(* IEC 61131-3 sources: smart-traffic-light/src/FunctionBlocks, 5 files *)

(* ---- PedestrianLight.st ---- *)
(* PedestrianLight Function Block
   Extends TrafficLight with pedestrian signal logic.
   Manages WALK/DONT_WALK/FLASHING states coordinated with the traffic signal. *)

FUNCTION_BLOCK PedestrianLight EXTENDS TrafficLight
  VAR_INPUT
    walkRequest  : BOOL := FALSE;
    walkDuration : TIME := T#20s;
  END_VAR

  VAR_OUTPUT
    pedestrianState : PedestrianState := PedestrianState.DONT_WALK;
    walkLight       : BOOL := FALSE;
    dontWalkLight   : BOOL := TRUE;
  END_VAR

  VAR
    walkTimer      : TON;
    flashTimer     : TON;
    flashCount     : INT := 0;
    maxFlashes     : INT := 5;
    flashOn        : BOOL := FALSE;
  END_VAR

  METHOD PUBLIC OVERRIDE GetState : TrafficState
    GetState := currentState;
  END_METHOD

  METHOD PUBLIC IsWalking : BOOL
    IsWalking := (pedestrianState = PedestrianState.WALK);
  END_METHOD

  METHOD PUBLIC RequestWalk : BOOL
    walkRequest := TRUE;
    RequestWalk := TRUE;
  END_METHOD

  (* Execute parent TrafficLight state machine first *)
  SUPER^();

  (* Pedestrian signal logic coordinated with traffic state *)
  IF currentState = TrafficState.RED AND walkRequest THEN
    (* Safe to walk when traffic is RED *)
    IF pedestrianState = PedestrianState.DONT_WALK THEN
      pedestrianState := PedestrianState.WALK;
      flashCount := 0;
    END_IF;

    walkTimer(IN := (pedestrianState = PedestrianState.WALK), PT := walkDuration);

    IF walkTimer.Q THEN
      pedestrianState := PedestrianState.FLASHING;
      walkTimer(IN := FALSE, PT := walkDuration);
    END_IF;

    (* Flashing phase before switching to DONT_WALK *)
    IF pedestrianState = PedestrianState.FLASHING THEN
      flashTimer(IN := TRUE, PT := T#500ms);
      IF flashTimer.Q THEN
        flashCount := flashCount + 1;
        flashOn := NOT flashOn;
        flashTimer(IN := FALSE, PT := T#500ms);
        flashTimer(IN := TRUE, PT := T#500ms);
      END_IF;

      IF flashCount >= maxFlashes THEN
        pedestrianState := PedestrianState.DONT_WALK;
        walkRequest := FALSE;
        flashCount := 0;
        flashOn := FALSE;
      END_IF;
    END_IF;
  ELSE
    (* Not safe or not requested — reset to DONT_WALK *)
    IF currentState <> TrafficState.RED THEN
      walkRequest := FALSE;
    END_IF;
    pedestrianState := PedestrianState.DONT_WALK;
    flashCount := 0;
    flashOn := FALSE;
    (* Reset timers to prevent stale state on next walk cycle *)
    walkTimer(IN := FALSE, PT := walkDuration);
    flashTimer(IN := FALSE, PT := T#500ms);
  END_IF;

  (* Update pedestrian signal outputs *)
  walkLight := (pedestrianState = PedestrianState.WALK) OR
               (pedestrianState = PedestrianState.FLASHING AND flashOn);
  dontWalkLight := (pedestrianState = PedestrianState.DONT_WALK) OR
                   (pedestrianState = PedestrianState.FLASHING AND NOT flashOn);
END_FUNCTION_BLOCK

(* ---- TrafficLight.st ---- *)
(* TrafficLight Function Block
   State machine for a standard 3-phase traffic signal.
   Cycles: RED -> GREEN -> YELLOW -> RED
   Supports night mode with flashing yellow. *)

FUNCTION_BLOCK TrafficLight IMPLEMENTS IControllable
  VAR_INPUT
    active    : BOOL := TRUE;
    timing    : PhaseTiming;
    nightMode : BOOL := FALSE;
  END_VAR

  VAR_OUTPUT
    currentState : TrafficState := TrafficState.RED;
    redLight     : BOOL := TRUE;
    yellowLight  : BOOL := FALSE;
    greenLight   : BOOL := FALSE;
  END_VAR

  VAR
    phaseTimer      : TON;
    flashTimer      : TON;
    currentDuration : TIME;
    flashOn         : BOOL := FALSE;
  END_VAR

  METHOD PUBLIC GetState : TrafficState
    GetState := currentState;
  END_METHOD

  METHOD PUBLIC IsGreen : BOOL
    IsGreen := (currentState = TrafficState.GREEN);
  END_METHOD

  METHOD PUBLIC IsRed : BOOL
    IsRed := (currentState = TrafficState.RED);
  END_METHOD

  METHOD PUBLIC IsNightMode : BOOL
    IsNightMode := nightMode;
  END_METHOD

  (* IControllable interface methods *)
  METHOD PUBLIC Enable : BOOL
    active := TRUE;
    Enable := TRUE;
  END_METHOD

  METHOD PUBLIC Disable : BOOL
    active := FALSE;
    Disable := TRUE;
  END_METHOD

  METHOD PUBLIC IsEnabled : BOOL
    IsEnabled := active;
  END_METHOD

  METHOD PUBLIC GetStatus : INT
    (* Status codes: 0=disabled, 1=RED, 2=GREEN, 3=YELLOW, 4=night mode *)
    IF NOT active THEN
      GetStatus := 0;
    ELSIF nightMode THEN
      GetStatus := 4;
    ELSIF currentState = TrafficState.RED THEN
      GetStatus := 1;
    ELSIF currentState = TrafficState.GREEN THEN
      GetStatus := 2;
    ELSE
      GetStatus := 3;
    END_IF;
  END_METHOD

  IF nightMode THEN
    (* Night mode: flash yellow at 1Hz *)
    flashTimer(IN := TRUE, PT := T#500ms);
    IF flashTimer.Q THEN
      flashOn := NOT flashOn;
      flashTimer(IN := FALSE, PT := T#500ms);
      flashTimer(IN := TRUE, PT := T#500ms);
    END_IF;

    redLight    := FALSE;
    yellowLight := flashOn;
    greenLight  := FALSE;
    currentState := TrafficState.YELLOW;
  ELSE
    (* Normal operation *)
    flashOn := FALSE;

    (* Determine the duration for the current phase *)
    CASE currentState OF
      TrafficState.RED:
        currentDuration := timing.redDuration;
      TrafficState.GREEN:
        currentDuration := timing.greenDuration;
      TrafficState.YELLOW:
        currentDuration := timing.yellowDuration;
    END_CASE;

    (* Run the phase timer *)
    phaseTimer(IN := active, PT := currentDuration);

    (* Transition to the next state when timer expires *)
    IF phaseTimer.Q THEN
      CASE currentState OF
        TrafficState.RED:
          currentState := TrafficState.GREEN;
        TrafficState.GREEN:
          currentState := TrafficState.YELLOW;
        TrafficState.YELLOW:
          currentState := TrafficState.RED;
      END_CASE;
      (* Reset timer for next phase *)
      phaseTimer(IN := FALSE, PT := currentDuration);
      phaseTimer(IN := active, PT := currentDuration);
    END_IF;

    (* Update output lights based on current state *)
    redLight    := (currentState = TrafficState.RED);
    yellowLight := (currentState = TrafficState.YELLOW);
    greenLight  := (currentState = TrafficState.GREEN);
  END_IF;
END_FUNCTION_BLOCK

(* ---- TrafficLogger.st ---- *)
(* TrafficLogger Function Block
   Maintains a circular buffer of state transition log entries.
   Uses dynamic memory allocation for the log buffer. *)

FUNCTION_BLOCK TrafficLogger
  VAR_INPUT
    bufferSize : INT := 20;
  END_VAR

  VAR_OUTPUT
    entryCount : INT := 0;
    isFull     : BOOL := FALSE;
  END_VAR

  VAR
    logBuffer    : POINTER TO LogEntry;
    writeIndex   : INT := 0;
    initialized  : BOOL := FALSE;
    totalEntries : DINT := 0;
  END_VAR

  METHOD PUBLIC Initialize : BOOL
    IF NOT initialized THEN
      logBuffer := __NEW(LogEntry, bufferSize);
      initialized := TRUE;
      Initialize := TRUE;
    ELSE
      Initialize := FALSE;
    END_IF;
  END_METHOD

  METHOD PUBLIC Cleanup : BOOL
    IF initialized THEN
      __DELETE(logBuffer);
      initialized := FALSE;
      entryCount := 0;
      writeIndex := 0;
      totalEntries := 0;
      isFull := FALSE;
      Cleanup := TRUE;
    ELSE
      Cleanup := FALSE;
    END_IF;
  END_METHOD

  METHOD PUBLIC LogTransition : BOOL
    VAR_INPUT
      fromState : TrafficState;
      toState   : TrafficState;
      time      : TIME;
    END_VAR

    IF NOT initialized THEN
      LogTransition := FALSE;
      RETURN;
    END_IF;

    logBuffer[writeIndex].previousState := fromState;
    logBuffer[writeIndex].newState := toState;
    logBuffer[writeIndex].timestamp := time;

    writeIndex := writeIndex + 1;
    IF writeIndex >= bufferSize THEN
      writeIndex := 0;
      isFull := TRUE;
    END_IF;

    totalEntries := totalEntries + 1;

    IF entryCount < bufferSize THEN
      entryCount := entryCount + 1;
    END_IF;

    LogTransition := TRUE;
  END_METHOD

  METHOD PUBLIC GetTotalTransitions : DINT
    GetTotalTransitions := totalEntries;
  END_METHOD
END_FUNCTION_BLOCK

(* ---- TurnSignalLight.st ---- *)
(* TurnSignalLight Function Block
   Extends TrafficLight with a dedicated turn signal arrow.
   The turn arrow activates during the RED-to-GREEN transition. *)

FUNCTION_BLOCK TurnSignalLight EXTENDS TrafficLight
  VAR_INPUT
    turnEnabled   : BOOL := TRUE;
    turnDuration  : TIME := T#10s;
  END_VAR

  VAR_OUTPUT
    turnArrowOn   : BOOL := FALSE;
    turnDirection : INT := 0;   (* 0=none, 1=left, 2=right *)
  END_VAR

  VAR
    turnTimer    : TON;
    turnActive   : BOOL := FALSE;
    prevState    : TrafficState := TrafficState.RED;
  END_VAR

  METHOD PUBLIC SetLeftTurn : BOOL
    turnDirection := 1;
    SetLeftTurn := TRUE;
  END_METHOD

  METHOD PUBLIC SetRightTurn : BOOL
    turnDirection := 2;
    SetRightTurn := TRUE;
  END_METHOD

  METHOD PUBLIC IsTurnActive : BOOL
    IsTurnActive := turnArrowOn;
  END_METHOD

  (* Run parent TrafficLight state machine first *)
  SUPER^();

  (* Detect RED-to-GREEN transition to activate turn signal *)
  IF prevState = TrafficState.RED AND currentState = TrafficState.GREEN THEN
    IF turnEnabled AND turnDirection > 0 THEN
      turnActive := TRUE;
    END_IF;
  END_IF;

  (* Run turn signal timer *)
  turnTimer(IN := turnActive, PT := turnDuration);
  IF turnTimer.Q THEN
    turnActive := FALSE;
    turnTimer(IN := FALSE, PT := turnDuration);
  END_IF;

  (* Turn off arrow when not in GREEN phase *)
  IF currentState <> TrafficState.GREEN THEN
    turnActive := FALSE;
  END_IF;

  turnArrowOn := turnActive;
  prevState := currentState;
END_FUNCTION_BLOCK

(* ---- VehicleDetector.st ---- *)
(* VehicleDetector Function Block
   Detects vehicles using a sensor input and maintains a detection history
   buffer allocated with dynamic memory. *)

FUNCTION_BLOCK VehicleDetector
  VAR_INPUT
    sensorInput   : BOOL := FALSE;
    maxHistory    : INT := 10;
  END_VAR

  VAR_OUTPUT
    vehicleCount  : INT := 0;
    isOccupied    : BOOL := FALSE;
    lastDetected  : TIME := T#0s;
  END_VAR

  VAR
    prevSensor     : BOOL := FALSE;
    historyBuffer  : POINTER TO INT;
    historySize    : INT := 0;
    initialized    : BOOL := FALSE;
    currentTime    : TIME := T#0s;
  END_VAR

  METHOD PUBLIC Initialize : BOOL
    IF NOT initialized THEN
      historyBuffer := __NEW(INT, maxHistory);
      initialized := TRUE;
      Initialize := TRUE;
    ELSE
      Initialize := FALSE;
    END_IF;
  END_METHOD

  METHOD PUBLIC Cleanup : BOOL
    IF initialized THEN
      __DELETE(historyBuffer);
      initialized := FALSE;
      historySize := 0;
      Cleanup := TRUE;
    ELSE
      Cleanup := FALSE;
    END_IF;
  END_METHOD

  METHOD PUBLIC GetDetectionCount : INT
    GetDetectionCount := vehicleCount;
  END_METHOD

  METHOD PUBLIC Reset : BOOL
    vehicleCount := 0;
    historySize := 0;
    isOccupied := FALSE;
    Reset := TRUE;
  END_METHOD

  (* Rising edge detection — count new vehicles *)
  IF sensorInput AND NOT prevSensor THEN
    vehicleCount := vehicleCount + 1;
    isOccupied := TRUE;
    lastDetected := currentTime;
  END_IF;

  IF NOT sensorInput AND prevSensor THEN
    isOccupied := FALSE;
  END_IF;

  prevSensor := sensorInput;
END_FUNCTION_BLOCK
